GLOBALCONSTANTS SubStrings (* Global constants *)
  (* Standard: 61499-1 *)
  (* Version 1.0, 2026-08-30, Franz Höpfinger, Meisterschulen am Ostbahnhof *)
  PACKAGE Meins::InputOutputTester::Button_PI_OPC_UA;
  VAR_GLOBAL CONSTANT
    PI_I1_COUNT_WRITE : WSTRING := "opc_ua[WRITE;/Objects/Pulse/I1/COUNT,1:s=PI_I1_COUNT]";
    PI_I1_FREQ_WRITE : WSTRING := "opc_ua[WRITE;/Objects/Pulse/I1/FREQ,1:s=PI_I1_FREQ]";
    PI_I1_SWITCH_READ : WSTRING := "opc_ua[READ;/Objects/Pulse/I1/SWITCH,1:s=PI_I1_SWITCH]";
    PI_I1_SWITCH_WRITE : WSTRING := "opc_ua[WRITE;/Objects/Pulse/I1/SWITCH,1:s=PI_I1_SWITCH]";
    PI_I1_STATUS_WRITE : WSTRING := "opc_ua[WRITE;/Objects/Pulse/I1/STATUS,1:s=PI_I1_STATUS]";
    PI_I2_COUNT_WRITE : WSTRING := "opc_ua[WRITE;/Objects/Pulse/I2/COUNT,1:s=PI_I2_COUNT]";
    PI_I2_FREQ_WRITE : WSTRING := "opc_ua[WRITE;/Objects/Pulse/I2/FREQ,1:s=PI_I2_FREQ]";
    PI_I2_SWITCH_READ : WSTRING := "opc_ua[READ;/Objects/Pulse/I2/SWITCH,1:s=PI_I2_SWITCH]";
    PI_I2_SWITCH_WRITE : WSTRING := "opc_ua[WRITE;/Objects/Pulse/I2/SWITCH,1:s=PI_I2_SWITCH]";
    PI_I2_STATUS_WRITE : WSTRING := "opc_ua[WRITE;/Objects/Pulse/I2/STATUS,1:s=PI_I2_STATUS]";
    PI_I3_COUNT_WRITE : WSTRING := "opc_ua[WRITE;/Objects/Pulse/I3/COUNT,1:s=PI_I3_COUNT]";
    PI_I3_FREQ_WRITE : WSTRING := "opc_ua[WRITE;/Objects/Pulse/I3/FREQ,1:s=PI_I3_FREQ]";
    PI_I3_SWITCH_READ : WSTRING := "opc_ua[READ;/Objects/Pulse/I3/SWITCH,1:s=PI_I3_SWITCH]";
    PI_I3_SWITCH_WRITE : WSTRING := "opc_ua[WRITE;/Objects/Pulse/I3/SWITCH,1:s=PI_I3_SWITCH]";
    PI_I3_STATUS_WRITE : WSTRING := "opc_ua[WRITE;/Objects/Pulse/I3/STATUS,1:s=PI_I3_STATUS]";
    PI_I4_COUNT_WRITE : WSTRING := "opc_ua[WRITE;/Objects/Pulse/I4/COUNT,1:s=PI_I4_COUNT]";
    PI_I4_FREQ_WRITE : WSTRING := "opc_ua[WRITE;/Objects/Pulse/I4/FREQ,1:s=PI_I4_FREQ]";
    PI_I4_SWITCH_READ : WSTRING := "opc_ua[READ;/Objects/Pulse/I4/SWITCH,1:s=PI_I4_SWITCH]";
    PI_I4_SWITCH_WRITE : WSTRING := "opc_ua[WRITE;/Objects/Pulse/I4/SWITCH,1:s=PI_I4_SWITCH]";
    PI_I4_STATUS_WRITE : WSTRING := "opc_ua[WRITE;/Objects/Pulse/I4/STATUS,1:s=PI_I4_STATUS]";
    PI_I5_COUNT_WRITE : WSTRING := "opc_ua[WRITE;/Objects/Pulse/I5/COUNT,1:s=PI_I5_COUNT]";
    PI_I5_FREQ_WRITE : WSTRING := "opc_ua[WRITE;/Objects/Pulse/I5/FREQ,1:s=PI_I5_FREQ]";
    PI_I5_SWITCH_READ : WSTRING := "opc_ua[READ;/Objects/Pulse/I5/SWITCH,1:s=PI_I5_SWITCH]";
    PI_I5_SWITCH_WRITE : WSTRING := "opc_ua[WRITE;/Objects/Pulse/I5/SWITCH,1:s=PI_I5_SWITCH]";
    PI_I5_STATUS_WRITE : WSTRING := "opc_ua[WRITE;/Objects/Pulse/I5/STATUS,1:s=PI_I5_STATUS]";
    PI_I6_COUNT_WRITE : WSTRING := "opc_ua[WRITE;/Objects/Pulse/I6/COUNT,1:s=PI_I6_COUNT]";
    PI_I6_FREQ_WRITE : WSTRING := "opc_ua[WRITE;/Objects/Pulse/I6/FREQ,1:s=PI_I6_FREQ]";
    PI_I6_SWITCH_READ : WSTRING := "opc_ua[READ;/Objects/Pulse/I6/SWITCH,1:s=PI_I6_SWITCH]";
    PI_I6_SWITCH_WRITE : WSTRING := "opc_ua[WRITE;/Objects/Pulse/I6/SWITCH,1:s=PI_I6_SWITCH]";
    PI_I6_STATUS_WRITE : WSTRING := "opc_ua[WRITE;/Objects/Pulse/I6/STATUS,1:s=PI_I6_STATUS]";
    PI_I7_COUNT_WRITE : WSTRING := "opc_ua[WRITE;/Objects/Pulse/I7/COUNT,1:s=PI_I7_COUNT]";
    PI_I7_FREQ_WRITE : WSTRING := "opc_ua[WRITE;/Objects/Pulse/I7/FREQ,1:s=PI_I7_FREQ]";
    PI_I7_SWITCH_READ : WSTRING := "opc_ua[READ;/Objects/Pulse/I7/SWITCH,1:s=PI_I7_SWITCH]";
    PI_I7_SWITCH_WRITE : WSTRING := "opc_ua[WRITE;/Objects/Pulse/I7/SWITCH,1:s=PI_I7_SWITCH]";
    PI_I7_STATUS_WRITE : WSTRING := "opc_ua[WRITE;/Objects/Pulse/I7/STATUS,1:s=PI_I7_STATUS]";
    PI_I8_COUNT_WRITE : WSTRING := "opc_ua[WRITE;/Objects/Pulse/I8/COUNT,1:s=PI_I8_COUNT]";
    PI_I8_FREQ_WRITE : WSTRING := "opc_ua[WRITE;/Objects/Pulse/I8/FREQ,1:s=PI_I8_FREQ]";
    PI_I8_SWITCH_READ : WSTRING := "opc_ua[READ;/Objects/Pulse/I8/SWITCH,1:s=PI_I8_SWITCH]";
    PI_I8_SWITCH_WRITE : WSTRING := "opc_ua[WRITE;/Objects/Pulse/I8/SWITCH,1:s=PI_I8_SWITCH]";
    PI_I8_STATUS_WRITE : WSTRING := "opc_ua[WRITE;/Objects/Pulse/I8/STATUS,1:s=PI_I8_STATUS]";
    Q01_READ : WSTRING := "opc_ua[READ;/Objects/DigitalOutput/Q01,1:s=Q01]";
    Q01_WRITE : WSTRING := "opc_ua[WRITE;/Objects/DigitalOutput/Q01,1:s=Q01]";
    Q02_READ : WSTRING := "opc_ua[READ;/Objects/DigitalOutput/Q02,1:s=Q02]";
    Q02_WRITE : WSTRING := "opc_ua[WRITE;/Objects/DigitalOutput/Q02,1:s=Q02]";
    Q03_READ : WSTRING := "opc_ua[READ;/Objects/DigitalOutput/Q03,1:s=Q03]";
    Q03_WRITE : WSTRING := "opc_ua[WRITE;/Objects/DigitalOutput/Q03,1:s=Q03]";
    Q04_READ : WSTRING := "opc_ua[READ;/Objects/DigitalOutput/Q04,1:s=Q04]";
    Q04_WRITE : WSTRING := "opc_ua[WRITE;/Objects/DigitalOutput/Q04,1:s=Q04]";
    Q05_READ : WSTRING := "opc_ua[READ;/Objects/DigitalOutput/Q05,1:s=Q05]";
    Q05_WRITE : WSTRING := "opc_ua[WRITE;/Objects/DigitalOutput/Q05,1:s=Q05]";
    Q06_READ : WSTRING := "opc_ua[READ;/Objects/DigitalOutput/Q06,1:s=Q06]";
    Q06_WRITE : WSTRING := "opc_ua[WRITE;/Objects/DigitalOutput/Q06,1:s=Q06]";
    Q07_READ : WSTRING := "opc_ua[READ;/Objects/DigitalOutput/Q07,1:s=Q07]";
    Q07_WRITE : WSTRING := "opc_ua[WRITE;/Objects/DigitalOutput/Q07,1:s=Q07]";
    Q08_READ : WSTRING := "opc_ua[READ;/Objects/DigitalOutput/Q08,1:s=Q08]";
    Q08_WRITE : WSTRING := "opc_ua[WRITE;/Objects/DigitalOutput/Q08,1:s=Q08]";
    Q09_READ : WSTRING := "opc_ua[READ;/Objects/DigitalOutput/Q09,1:s=Q09]";
    Q09_WRITE : WSTRING := "opc_ua[WRITE;/Objects/DigitalOutput/Q09,1:s=Q09]";
    Q10_READ : WSTRING := "opc_ua[READ;/Objects/DigitalOutput/Q10,1:s=Q10]";
    Q10_WRITE : WSTRING := "opc_ua[WRITE;/Objects/DigitalOutput/Q10,1:s=Q10]";
    Q11_READ : WSTRING := "opc_ua[READ;/Objects/DigitalOutput/Q11,1:s=Q11]";
    Q11_WRITE : WSTRING := "opc_ua[WRITE;/Objects/DigitalOutput/Q11,1:s=Q11]";
    Q12_READ : WSTRING := "opc_ua[READ;/Objects/DigitalOutput/Q12,1:s=Q12]";
    Q12_WRITE : WSTRING := "opc_ua[WRITE;/Objects/DigitalOutput/Q12,1:s=Q12]";
    Tick_WRITE : WSTRING := "opc_ua[WRITE;/Objects/System/Tick,1:s=System.Tick]";
  END_VAR
END_GLOBALCONSTANTS
